FUNCTION F_DebugCompositionCustomization : BOOL



(****************************************************************************************
   Add custom code that shall be executed during debug here.
*****************************************************************************************)
;


(****************************************************************************************
   Example: Configure project when running Demo3D simulator
*****************************************************************************************)
IF(DEMO3D_SIM_ENABLED) THEN
	;
	(*
	Groups.fbSG_001.HW_Inputs.AutoOnPB 						:= TRUE;
	Groups.fbSG_001.HW_Inputs.EmergencyCircuitOK 			:= TRUE;
	Groups.fbSG_001.HW_Inputs.ManAutoSW 					:= TRUE;
	Groups.fbSG_001.HW_Inputs.ResetErrorPB 					:= ResetErrorSG1; 
	Groups.fbSG_001.HW_Inputs.MainContactorOFF				:= TRUE; 
	Groups.fbSG_001.HW_Inputs.FeedbackMainContactorOFF[1]	:= TRUE; 
	Groups.fbSG_001.HW_Inputs.FeedbackMainContactorOFF[2]	:= TRUE; 
	Groups.fbSG_001.HW_Inputs.FeedbackMainContactorOFF[3]	:= TRUE; 
	Groups.fbSG_001.HW_Inputs.FeedbackMainContactorOFF[4]	:= TRUE; 
	Groups.fbSG_001.HW_Inputs.FireAlarm						:= TRUE; 
	*)
END_IF

END_FUNCTION

(* stored: Version 1.1.0.1, ProductVersion 3.1.4024.9
   POU F_DebugCompositionCustomization: Id {bdd2a976-368f-41f7-a5e3-f6d769339915}, SpecialFunc None *)
